// TIA Portal project "FactoryIO_Template_S7-1200_V16_V16" (V16)
// Vorlageprojekt für das Buch mit Zielsystem S7-1200

(* hardware
DEVICE "S7-1200-Station_1"  S7-1200 Station
   slot 0: "Baugruppenträger_0"  Rack  V1.0
   slot 1: "PLC_1"  CPU 1211C DC/DC/DC  6ES7 211-1AE40-0XB0  V4.1
*)

// ===== PLC "PLC_1"  CPU 1211C DC/DC/DC =====

VAR_GLOBAL   // PLC tag table "Standard-Variablentabelle"
   "START" AT %I0.0 : Bool;
   "STOP" AT %I0.1 : Bool;
   "SMALL SENSOR" AT %I0.2 : Bool;
   "HIGH SENSOR" AT %I0.3 : Bool;
   "TWO AXIS SENSOR" AT %I0.4 : Bool;
   "MOVING X" AT %I0.5 : Bool;
   "MOVING Z" AT %I0.6 : Bool;
   "EMITTER" AT %Q0.0 : Bool;
   "ENTRY" AT %Q0.1 : Bool;
   "SORTING" AT %Q0.2 : Bool;
   "SMALL" AT %Q0.3 : Bool;
   "LARGE" AT %Q0.4 : Bool;
   "X" AT %Q0.5 : Bool;
   "Z" AT %Q0.6 : Bool;
   "GRAB" AT %Q0.7 : Bool;
   "CW" AT %Q1.0 : Bool;
   "CCW" AT %Q1.1 : Bool;
   "MARKER 1" AT %M0.1 : Bool;
   "MARKER 2" AT %M0.2 : Bool;
   "MARKER 3" AT %M0.3 : Bool;
   "MARKER 4" AT %M0.4 : Bool;
   "MARKER 5" AT %M0.5 : Bool;
   "DETECTED" AT %I0.7 : Bool;
   "ROTATING" AT %I1.0 : Bool;
   "MARKER 6" AT %M0.6 : Bool;
   "MARKER 7" AT %M0.7 : Bool;
   "MARKER 8" AT %M1.0 : Bool;
   "MARKER 9" AT %M1.1 : Bool;
   "MARKER 10" AT %M1.2 : Bool;
END_VAR

// folder: System blocks/Program resources

DATA_BLOCK "C1"   // DB1
{ S7_Optimized_Access := 'TRUE' }
AUTHOR : Simatic
FAMILY : IEC
NAME : CNTR
VERSION : 1.0
// stored: InstanceOfName IEC_COUNTER
"IEC_COUNTER"
BEGIN
END_DATA_BLOCK

// folder: (top level)

FUNCTION "MHJ-PLC-Lab-Function-S71200" : Void   // FC9000, SCL
{ S7_Optimized_Access := 'TRUE' }
VERSION : 0.1
   VAR_TEMP
      rdTimeReturn : Int;
      outputTime : DTL;
      SyncVal : Byte;
      forVal : Int;
      forVal_2 : Int;
      Value : Byte;
   END_VAR
   VAR CONSTANT
      CompVal : Byte := 16#34;
      Value_01 : Byte := 16#11;
      Value_01_DW : DWord := 16#A165_D992;
      Value_02_DW : DWord := 16#58BE_4401;
   END_VAR
BEGIN

   #Value:=PEEK(area := 16#82,
        dbNumber := 0,
        byteOffset := 511);
   #Value := #Value + 1;

   POKE(area := 16#82,
        dbNumber := 0,
        byteOffset := 511,
        value := #Value);

   POKE(area:=16#81,
        dbNumber:=0,
        byteOffset:=1016,
        value:=#Value_01_DW);
   POKE(area := 16#81,
        dbNumber := 0,
        byteOffset := 1020,
        value := #Value_02_DW);

   POKE(area := 16#81,
        dbNumber := 0,
        byteOffset := 511,
        value := B#16#00);

   FOR #forVal := 0 TO 120 DO
       FOR #forVal_2:=0 TO 10 DO
           #rdTimeReturn:=RD_SYS_T(#outputTime);
           #rdTimeReturn := WR_SYS_T(#outputTime);
           #rdTimeReturn := RD_SYS_T(#outputTime);
           #rdTimeReturn := WR_SYS_T(#outputTime);
       END_FOR;
       #SyncVal:= PEEK(area := 16#81,
                      dbNumber := 0,
                      byteOffset := 511);
       IF #SyncVal = #CompVal THEN
          GOTO M_1;
       END_IF;
   END_FOR;
   RETURN;

   M_1:
   POKE(area := 16#81,
        dbNumber := 0,
        byteOffset := 511,
        value := B#16#0);
END_FUNCTION

ORGANIZATION_BLOCK "Main"   // OB1, LAD, ProgramCycle
TITLE = "Main Program Sweep (Cycle)"
{ S7_Optimized_Access := 'TRUE' }
VERSION : 0.1
   VAR_INPUT
      Initial_Call : Bool;   // Initial call of this OB
      Remanence : Bool;   // =True, if remanent data are available
   END_VAR
   VAR_TEMP   // added for the SCL form of the ladder/FBD networks
      _w1 : Bool;
      _w2 : Bool;
      _w3 : Bool;
      _w4 : Bool;
   END_VAR
BEGIN

REGION Network 1: Konnektierungsbaustein für PLC-Lab
   // Im Netzwerk 1 wird der Konnektierungsbaustein für PLC-Lab aufgerufen.
   // Dieser Aufruf darf nicht entfernt werden!
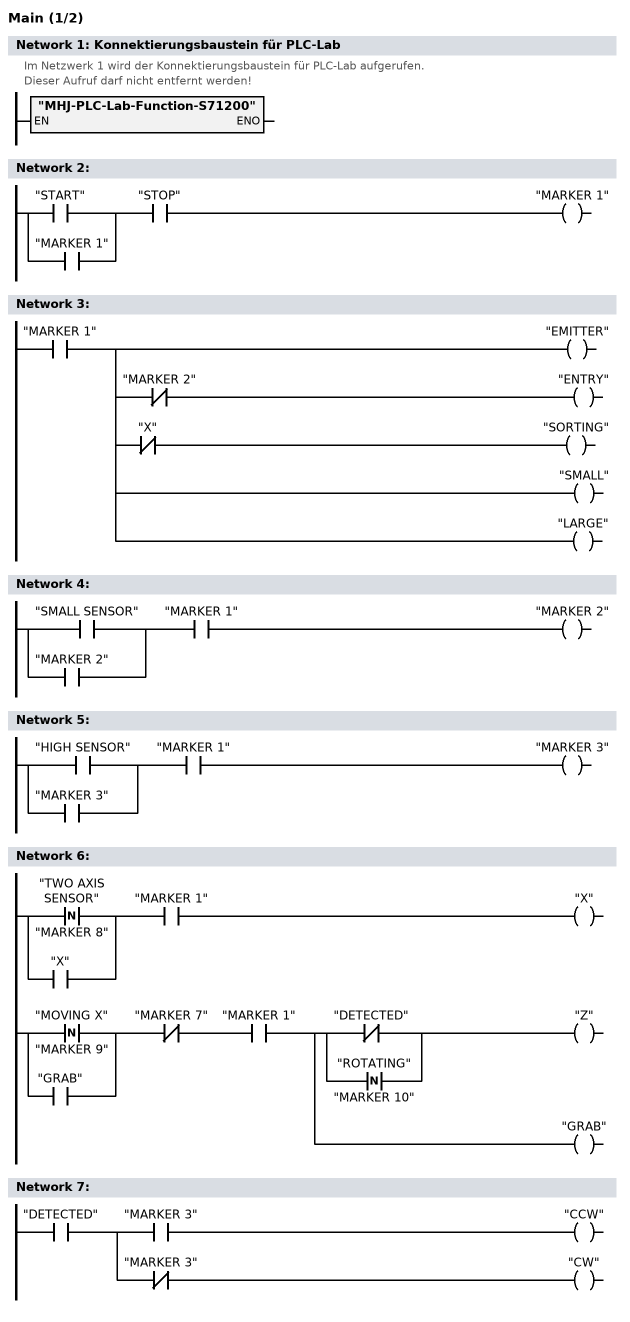
   RUNG wire#powerrail
      "MHJ-PLC-Lab-Function-S71200"()
   END_RUNG
   // the same network as SCL:
   "MHJ-PLC-Lab-Function-S71200"();
END_REGION

REGION Network 2
   RUNG wire#powerrail
      Contact( "START" )
      wire#w1
      Contact( "STOP" )
      Coil( "MARKER 1" )
   END_RUNG
   RUNG wire#powerrail
      Contact( "MARKER 1" )
   END_RUNG wire#w1
   // the same network as SCL:
   "MARKER 1" := ("START" OR "MARKER 1") AND "STOP";
END_REGION

REGION Network 3
   RUNG wire#powerrail
      Contact( "MARKER 1" )
      wire#w1
      Coil( "EMITTER" )
   END_RUNG
   RUNG wire#w1
      I_Contact( "MARKER 2" )
      Coil( "ENTRY" )
   END_RUNG
   RUNG wire#w1
      I_Contact( "X" )
      Coil( "SORTING" )
   END_RUNG
   RUNG wire#w1
      Coil( "SMALL" )
   END_RUNG
   RUNG wire#w1
      Coil( "LARGE" )
   END_RUNG
   // the same network as SCL:
   "EMITTER" := "MARKER 1";
   "ENTRY" := "MARKER 1" AND NOT "MARKER 2";
   "SORTING" := "MARKER 1" AND NOT "X";
   "SMALL" := "MARKER 1";
   "LARGE" := "MARKER 1";
END_REGION

REGION Network 4
   RUNG wire#powerrail
      Contact( "SMALL SENSOR" )
      wire#w1
      Contact( "MARKER 1" )
      Coil( "MARKER 2" )
   END_RUNG
   RUNG wire#powerrail
      Contact( "MARKER 2" )
   END_RUNG wire#w1
   // the same network as SCL:
   "MARKER 2" := ("SMALL SENSOR" OR "MARKER 2") AND "MARKER 1";
END_REGION

REGION Network 5
   RUNG wire#powerrail
      Contact( "HIGH SENSOR" )
      wire#w1
      Contact( "MARKER 1" )
      Coil( "MARKER 3" )
   END_RUNG
   RUNG wire#powerrail
      Contact( "MARKER 3" )
   END_RUNG wire#w1
   // the same network as SCL:
   "MARKER 3" := ("HIGH SENSOR" OR "MARKER 3") AND "MARKER 1";
END_REGION

REGION Network 6
   RUNG wire#powerrail
      N_Contact(operand := "TWO AXIS SENSOR", bit := "MARKER 8")
      wire#w1
      Contact( "MARKER 1" )
      Coil( "X" )
   END_RUNG
   RUNG wire#powerrail
      Contact( "X" )
   END_RUNG wire#w1
   RUNG wire#powerrail
      N_Contact(operand := "MOVING X", bit := "MARKER 9")
      wire#w2
      I_Contact( "MARKER 7" )
      Contact( "MARKER 1" )
      wire#w3
      I_Contact( "DETECTED" )
      wire#w4
      Coil( "Z" )
   END_RUNG
   RUNG wire#powerrail
      Contact( "GRAB" )
   END_RUNG wire#w2
   RUNG wire#w3
      N_Contact(operand := "ROTATING", bit := "MARKER 10")
   END_RUNG wire#w4
   RUNG wire#w3
      Coil( "GRAB" )
   END_RUNG
   // the same network as SCL:
   #_w1 := NOT "TWO AXIS SENSOR" AND "MARKER 8";   // falling edge of "TWO AXIS SENSOR"
   "MARKER 8" := "TWO AXIS SENSOR";
   "X" := (#_w1 OR "X") AND "MARKER 1";
   #_w2 := NOT "MOVING X" AND "MARKER 9";   // falling edge of "MOVING X"
   "MARKER 9" := "MOVING X";
   #_w3 := (#_w2 OR "GRAB") AND NOT "MARKER 7" AND "MARKER 1";
   #_w4 := #_w3 AND NOT "ROTATING" AND "MARKER 10";   // falling edge of "ROTATING"
   "MARKER 10" := "ROTATING";
   "Z" := (#_w3 AND NOT "DETECTED") OR #_w4;
   "GRAB" := #_w3;
END_REGION

REGION Network 7
   RUNG wire#powerrail
      Contact( "DETECTED" )
      wire#w1
      Contact( "MARKER 3" )
      Coil( "CCW" )
   END_RUNG
   RUNG wire#w1
      I_Contact( "MARKER 3" )
      Coil( "CW" )
   END_RUNG
   // the same network as SCL:
   "CCW" := "DETECTED" AND "MARKER 3";
   "CW" := "DETECTED" AND NOT "MARKER 3";
END_REGION

REGION Network 8
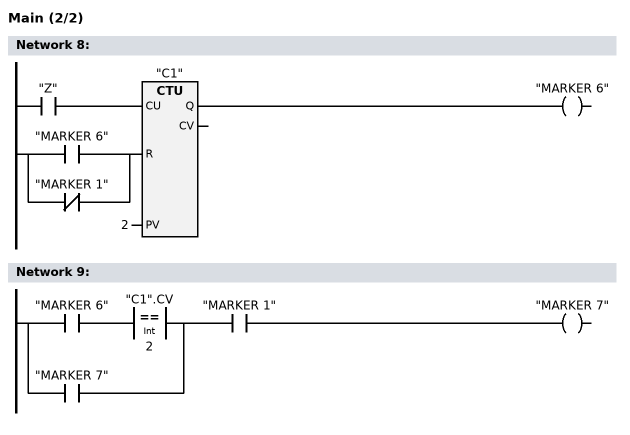
   "C1".CTU(CU := "Z", R := "MARKER 6" OR NOT "MARKER 1", PV := 2);
   "MARKER 6" := "C1".Q;
END_REGION

REGION Network 9
   RUNG wire#powerrail
      Contact( "MARKER 6" )
      { S7_Templates := "SrcType := Int" } EQ_Contact(in1 := "C1".CV, in2 := 2)
      wire#w1
      Contact( "MARKER 1" )
      Coil( "MARKER 7" )
   END_RUNG
   RUNG wire#powerrail
      Contact( "MARKER 7" )
   END_RUNG wire#w1
   // the same network as SCL:
   "MARKER 7" := (("MARKER 6" AND ("C1".CV = 2)) OR "MARKER 7") AND "MARKER 1";
END_REGION
END_ORGANIZATION_BLOCK